(* PLC project CoDeSys External Library Template, WAGO e!COCKPIT e!COCKPIT, author 3S - Smart Software Solutions GmbH *)
(* stored: creationDateTime 2019-10-29T12:37:19.9513383, version 3.5.5.30, modificationDateTime 2019-10-29T12:36:39.3744516, organization 3S - Smart Software Solutions GmbH *)
(* Library project template with all possible element types, docu and a sample project structure *)

FUNCTION fnModbusZapisRejestru : BOOL
  VAR_INPUT
    bAdresUrzadzenia : BYTE;  (* ID urządzenia SLAVE w sieci MODBUS *)
    bFunkcja : BYTE;  (* kod funkcji użytej w rozkazie MODBUS *)
    uiAdresRejestru : UINT;  (* rejestr startowy *)
    pZmiennaReferencyjna : POINTER TO WORD;  (* wskaźnik do wartości do zapisu *)
    wWartoscDoZapisania : WORD;  (* wartość do zapisania *)
    intModbusOdczytZapisZadanieRozmiar : INT;
  END_VAR
  VAR_IN_OUT
    arModbusOdczytZapisZadanie : ARRAY[1..1000] OF typModbusOdczytZapisZadanie;
    intModbusOdczytZapisZadanieZnacznikZapisu : INT;
  END_VAR

            fnTablicaKomunikatowInkrementacja(intRozmiarTablicy := intModbusOdczytZapisZadanieRozmiar , intWskaznik := intModbusOdczytZapisZadanieZnacznikZapisu);

arModbusOdczytZapisZadanie[intModbusOdczytZapisZadanieZnacznikZapisu].bAdresUrzadzenia := bAdresUrzadzenia;
arModbusOdczytZapisZadanie[intModbusOdczytZapisZadanieZnacznikZapisu].bFunkcja := bFunkcja;
arModbusOdczytZapisZadanie[intModbusOdczytZapisZadanieZnacznikZapisu].uiAdresRejestru := uiAdresRejestru;
arModbusOdczytZapisZadanie[intModbusOdczytZapisZadanieZnacznikZapisu].pZmiennaDoOdczytu := pZmiennaReferencyjna;
arModbusOdczytZapisZadanie[intModbusOdczytZapisZadanieZnacznikZapisu].wWartoscDoZapisania := wWartoscDoZapisania;
          
END_FUNCTION
